// TIA Portal V17 export
// export: Created 2025-03-10T12:17:23.6832541Z, ExportSetting WithDefaults, DisplayName Totally Integrated Automation Portal, DisplayVersion V17 Update 8, DisplayName TIA Portal Openness, DisplayVersion V17 Update 8, DisplayName TIA Portal Version Control Interface, DisplayVersion V17, DisplayName SINAMICS Startdrive Advanced, DisplayVersion V17 SP2, DisplayName SINAMICS Startdrive G110M, G120, G120C, G120D, G120P, G115D, DisplayVersion V17 SP2, DisplayName SINAMICS Startdrive G130, G150, S120, S150, SINAMICS MV, S210, DisplayVersion V17 SP2, DisplayName STEP 7 Professional, DisplayVersion V17 Update 8, DisplayName SINUMERIK ONE STEP 7 Toolbox, DisplayVersion V17 Update 12, DisplayName SINUMERIK 840D sl STEP 7 Toolbox, DisplayVersion V17 Update 12, DisplayName STEP 7 Safety, DisplayVersion V17 Update 6, DisplayName WinCC Advanced, DisplayVersion V17 Update 8
DATA_BLOCK "DB7239_MULTIPLEX_VARIABLES"   // DB7239
{ S7_Optimized_Access := 'FALSE'; DB_Accessible_From_OPC_UA := 'FALSE' }
VERSION : 0.1
// stored: AutoNumber false, DBAccessibleFromOPCUA false, DBAccessibleFromWebserver true, IsOnlyStoredInLoadMemory false, IsWriteProtectedInAS false
   VAR
      VARIABLE_00 : Word;   // FIXTURE 1 PART STATUS
      VARIABLE_01 : Word;   // FIXTURE 2 PART STATUS
      VARIABLE_02 : Word;   // FIXTURE 3 PART STATUS
      VARIABLE_03 : Word;   // FIXTURE 4 PART STATUS
      VARIABLE_04 : Word;   // FIXTURE 1 PART QUALITY
      VARIABLE_05 : Word;   // FIXTURE 2 PART QUALITY
      VARIABLE_06 : Word;   // FIXTURE 3 PART QUALITY
      VARIABLE_07 : Word;   // FIXTURE 4 PART QUALITY
      VARIABLE_08 : Word;   // STATION 1 PART STATUS
      VARIABLE_09 : Word;   // STATION 2 PART STATUS
      VARIABLE_10 : Word;   // STATION 3 PART STATUS
      VARIABLE_11 : Word;   // STATION 4 PART STATUS
      VARIABLE_12 : Word;   // STATION 1 PART QUALITY
      VARIABLE_13 : Word;   // STATION 2 PART QUALITY
      VARIABLE_14 : Word;   // STATION 3 PART QUALITY
      VARIABLE_15 : Word;   // STATION 4 PART QUALITY
      VARIABLE_16 : Word;   // SPARE
      VARIABLE_17 : Word;   // SPARE
      VARIABLE_18 : Word;   // SPARE
      VARIABLE_19 : Word;   // SPARE
   END_VAR
BEGIN
END_DATA_BLOCK
